Staubli VAL3: strlength.pgx

program strlength(string& x_sMessage[], num x_nLength)
  local string lStrEmpty
  local string l_sTemp
begin
  lStrEmpty="                                        "
  // Look for asian message
  if getDisplayLen(x_sMessage)>x_nLength
    // Need to divide the message
    if getDisplayLen(x_sMessage)==len(x_sMessage)
      if mid(x_sMessage,1,x_nLength)!=" "
        // European message
        x_sMessage=mid(x_sMessage,x_nLength-1,0)
        x_sMessage=x_sMessage+"."
      else
        // Found and empty space
        x_sMessage=mid(x_sMessage,x_nLength,0)
      endIf
    else
      // Asian one
      call midPos(x_sMessage,x_nLength,0,x_sMessage)
    endIf
  else
    if getDisplayLen(x_sMessage)<x_nLength
      // European
      if getDisplayLen(x_sMessage)==len(x_sMessage)
        x_sMessage=x_sMessage+mid(lStrEmpty,x_nLength-getDisplayLen(x_sMessage),0)
      else
        // Asian
        call midPos(lStrEmpty,x_nLength-getDisplayLen(x_sMessage),0,l_sTemp)
        x_sMessage=x_sMessage+l_sTemp
      endIf
    else
      // They are the same
    endIf
  endIf
end
